{attribute 'linkalways'} 
{attribute 'no_explicit_call' := 'This FB is a CLASS and must be accessed using methods or properties'}
{attribute 'enable_dynamic_creation'}
FUNCTION_BLOCK _USINT EXTENDS NumericDatatypeBase
VAR
	localData : USINT;
	activeData : REFERENCE TO USINT REF= localData;
END_VAR

PROPERTY PUBLIC Address : PVOID
GET
Address := ADR(activeData);
END_GET
END_PROPERTY

METHOD PUBLIC ClearReference
VAR_INPUT
END_VAR
activeData REF= localData;
END_METHOD

METHOD PUBLIC Clone : I_Datatype
VAR
    pClone : POINTER TO _USINT;
END_VAR
pClone := __NEW(_USINT(InitialValue := Value));
Clone := pClone^;
END_METHOD

METHOD FB_init : BOOL
VAR_INPUT
	bInitRetains : BOOL; // if TRUE, the retain variables are initialized (warm start / cold start)
	bInCopyCode : BOOL;  // if TRUE, the instance afterwards gets moved into the copy code (online change)
	InitialValue : USINT;
END_VAR
localData := InitialValue;
END_METHOD

PROPERTY PUBLIC IsFloat : BOOL
GET
IsFloat := FALSE;
END_GET
END_PROPERTY

PROPERTY PUBLIC IsSigned : BOOL
GET
IsSigned := FALSE;
END_GET
END_PROPERTY

METHOD PUBLIC MakeReferenceTo
VAR_INPUT
	ReferenceTarget : REFERENCE TO USINT;
END_VAR
activeData REF= ReferenceTarget;
END_METHOD

PROPERTY PUBLIC MaxValue : USINT
GET
MaxValue :=  DatatypeLimits.USINT_MAX_VALUE;
END_GET
END_PROPERTY

PROPERTY PUBLIC MinValue : USINT
GET
MinValue := DatatypeLimits.USINT_MIN_VALUE;
END_GET
END_PROPERTY

METHOD PROTECTED SerializeMaxValue
VAR_INPUT
	Serializer : I_Serializer;
END_VAR
Serializer.AddUsint(MaxValue);
END_METHOD

METHOD PROTECTED SerializeMinValue
VAR_INPUT
	Serializer : I_Serializer;
END_VAR
Serializer.AddUsint(MinValue);
END_METHOD

METHOD PUBLIC SerializeWith
VAR_INPUT
	Serializer : I_Serializer;
END_VAR
Serializer.AddUsint(activeData);
END_METHOD

PROPERTY PUBLIC Size : UDINT
GET
Size := SIZEOF(activeData);
END_GET
END_PROPERTY

METHOD TryDeserializeFrom : BOOL
VAR_INPUT
	Deserializer : I_Deserializer;
	Feedback : I_DeserializerFeedback;
END_VAR
TryDeserializeFrom := Deserializer.TryGetUsint(activeData, Feedback);
END_METHOD

METHOD TryMakeReferenceTo : BOOL
VAR_INPUT
	Target : I_Datatype;
END_VAR
VAR
	pTargetData : POINTER TO USINT;
END_VAR
IF NOT (Target.TypeName = TypeName) THEN
	RETURN;
END_IF

pTargetData := Target.Address;
activeData REF= pTargetData^;
TryMakeReferenceTo := TRUE;
END_METHOD

PROPERTY PUBLIC TypeName : T_MAXSTRING
GET
TypeName := 'USINT';
END_GET
END_PROPERTY

PROPERTY PUBLIC Value : USINT
GET
Value := activeData;
END_GET
SET
activeData := Value;
END_SET
END_PROPERTY

END_FUNCTION_BLOCK

(* stored: Version 1.1.0.1, ProductVersion 3.1.4024.12
   POU _USINT: Id {c3b146d7-a462-0db1-3c7c-763f2ad2820b}, SpecialFunc None
   Folder Constructor: Id {5b67fd49-4685-053d-3c56-3c79816ef221}
   Folder Protected: Id {8904c364-edbc-0791-3b92-a05e5e446ab0}
   Property Address: Id {0449a95c-d8c1-00fa-2707-e2a0b87a5223}
   Get Get: Id {22e9dd9e-0c86-0d2d-3070-8579c619b567}
   Method ClearReference: Id {3a24a375-4c5d-0f9d-243e-dd8ed8334884}
   Method Clone: Id {2ee13ade-7167-0518-248d-7979a529cf4e}
   Method FB_init: Id {8e836f2e-fccb-0075-14fc-0281281bc71e}
   Property IsFloat: Id {c2c34d86-8085-040f-3f3a-9827cb9e3a41}
   Get Get: Id {bd410834-e394-0aa2-33ff-d48a8a6c3f3f}
   Property IsSigned: Id {8cbc6ceb-85bc-09a2-1f1c-84ffddbbbc9e}
   Get Get: Id {4d078ac3-58a5-0c36-1377-56065293577c}
   Method MakeReferenceTo: Id {276a0ea2-4a30-060b-332b-bcf23280dbef}
   Property MaxValue: Id {85daa3ae-9ed2-0367-26d4-0776e0964c15}
   Get Get: Id {346101bf-854f-0e3b-1f57-16093171e7ea}
   Property MinValue: Id {32a719f4-9486-035b-371b-89fb11e956d5}
   Get Get: Id {399ff623-1ec1-034e-0ec0-a470b5d5e944}
   Method SerializeMaxValue: Id {7da2e7b7-08e6-0b8a-3578-b1c50ce0635a}
   Method SerializeMinValue: Id {9792c06e-bc0a-083a-06d1-a7674f9a53c1}
   Method SerializeWith: Id {3320ec2d-ae10-03ad-3b96-5312a4debae2}
   Property Size: Id {a829dfd2-c970-024e-14f5-f58f5403ade7}
   Get Get: Id {75d712bf-887d-0b44-194c-21fe8b51dd15}
   Method TryDeserializeFrom: Id {6d2b7ef4-fd57-03de-21d6-38be9e9ddf64}
   Method TryMakeReferenceTo: Id {2d2c21cc-7403-0f5f-34d5-e28eef7a916e}
   Property TypeName: Id {46874b16-03e8-0876-32a5-38682ff67672}
   Get Get: Id {72cf7c21-f266-0fd7-2be9-37e19aa5041d}
   Property Value: Id {c795a587-8dc4-0fff-303e-5a8b8f9d8a3c}
   Get Get: Id {5ce174f7-9e17-0233-2c2c-a6eb59a52023}
   Set Set: Id {e73def83-567a-00c0-34ae-0e200ed35630} *)
